TYPE commUnitController EXTENDS commUnit :
STRUCT
	control : DWORD; //32
	errorIndex : DWORD; //34
	errorType : DWORD; //36
	errorCode : LWORD; // 38
	reserved2 : ARRAY[1..8] OF WORD;
	//monitorDatas : ARRAY[1..8] OF DWORD;
END_STRUCT
END_TYPE

(* stored: Version 1.1.0.1, ProductVersion 3.1.4022.10
   DUT commUnitController: Id {3540f8c1-cc91-4ec1-8a4f-7596595f2c82} *)
